// TIA Portal V16 export
// export: Created 2025-08-01T13:38:04.5785959Z, ExportSetting WithDefaults, DisplayName Totally Integrated Automation Portal, DisplayVersion V16, DisplayName TIA Portal Version Control Interface, DisplayVersion V16, DisplayName TIA Portal Openness, DisplayVersion V16, DisplayName STEP 7 Professional, DisplayVersion V16, DisplayName STEP 7 Safety, DisplayVersion V16, DisplayName WinCC Advanced, DisplayVersion V16
DATA_BLOCK "DB_EncoderBand"   // DB95
VERSION : 0.1
// stored: AutoNumber false, IsOnlyStoredInLoadMemory false, IsWriteProtectedInAS false
   VAR RETAIN
      ControlWord1 : DInt;
      ControlWord2 : DInt;
      FeedbackWord1 : DInt;
      FeedbackWord2 : DInt;
      EnableGate : Bool;
      ControlWord : Word;
      EncoderValue : DInt;
   END_VAR
BEGIN
END_DATA_BLOCK
